FUNCTION_BLOCK CountCurrentPosition1
VAR_INPUT
END_VAR
VAR_OUTPUT
END_VAR
VAR
END_VAR

// COUNT ROTATION:
IF IO.Initialized AND IO.StepRotatonSwitch = 1 THEN
	IF IO.MotorRotationDirection = 0 THEN
		IF (NOT IO.Switch) AND Automatic.RCurrentlyMoving THEN
			IF IO.PreviousManualMode THEN
				Automatic.RotationPositionCurrent := Automatic.RotationPositionCurrent + 1;
			ELSE
				Automatic.RotationPositionCurrent := Automatic.RotationPositionCurrent + 1;
				Automatic.RotationPositionAuto := Automatic.RotationPositionAuto + 1;
			END_IF
		ELSIF Automatic.RCurrentlyMoving THEN
			Automatic.RotationPositionCurrent := Automatic.RotationPositionCurrent + 1;
		END_IF
	ELSE
		IF (NOT IO.Switch) AND Automatic.RCurrentlyMoving THEN
			IF IO.PreviousManualMode THEN
				Automatic.RotationPositionCurrent := Automatic.RotationPositionCurrent - 1;
			ELSE
				Automatic.RotationPositionCurrent := Automatic.RotationPositionCurrent - 1;
				Automatic.RotationPositionAuto := Automatic.RotationPositionAuto - 1;
			END_IF
		ELSIF Automatic.RCurrentlyMoving THEN
			Automatic.RotationPositionCurrent := Automatic.RotationPositionCurrent - 1;
		END_IF
	END_IF
END_IF

// COUNT Extension:
IF IO.Initialized AND IO.StepExtensionSwitch = 1 THEN
	IO.LEDGreen := 0;
	IF IO.MotorExtensionDirection = 0 THEN
		IF (NOT IO.Switch) AND Automatic.ECurrentlyMoving THEN
			IF IO.PreviousManualMode THEN
				Automatic.ExtensionPositionCurrent := Automatic.ExtensionPositionCurrent + 1;
			ELSE
				Automatic.ExtensionPositionAuto := Automatic.ExtensionPositionAuto + 1;
				Automatic.ExtensionPositionCurrent := Automatic.ExtensionPositionCurrent + 1;
			END_IF
		ELSIF Automatic.ECurrentlyMoving THEN
			Automatic.ExtensionPositionCurrent := Automatic.ExtensionPositionCurrent + 1;
		END_IF
	ELSE
		IF (NOT IO.Switch) AND Automatic.ECurrentlyMoving THEN
			IF IO.PreviousManualMode THEN
				Automatic.ExtensionPositionCurrent := Automatic.ExtensionPositionCurrent - 1;
			ELSE
				Automatic.ExtensionPositionAuto := Automatic.ExtensionPositionAuto - 1;
				Automatic.ExtensionPositionCurrent := Automatic.ExtensionPositionCurrent - 1;
			END_IF
		ELSIF Automatic.ECurrentlyMoving THEN
			Automatic.ExtensionPositionCurrent := Automatic.ExtensionPositionCurrent - 1;
		END_IF
	END_IF
END_IF

// COUNT Lifting:
IF IO.Initialized AND IO.StepLiftingSwitch = 1 THEN
	IF IO.MotorLiftingDirection = 0 THEN
		IF (NOT IO.Switch) AND Automatic.LCurrentlyMoving THEN
			IF IO.PreviousManualMode THEN
				Automatic.LiftingPositionCurrent := Automatic.LiftingPositionCurrent + 1;
			ELSE
				Automatic.LiftingPositionCurrent := Automatic.LiftingPositionCurrent + 1;
				Automatic.LiftingPositionAuto := Automatic.LiftingPositionAuto + 1;
			END_IF
		ELSIF Automatic.LCurrentlyMoving THEN
			Automatic.LiftingPositionCurrent := Automatic.LiftingPositionCurrent + 1;
		END_IF
	ELSE
		IF (NOT IO.Switch) AND Automatic.LCurrentlyMoving THEN
			IF IO.PreviousManualMode THEN
				Automatic.LiftingPositionCurrent := Automatic.LiftingPositionCurrent - 1;
			ELSE
				Automatic.LiftingPositionAuto := Automatic.LiftingPositionAuto - 1;
				Automatic.LiftingPositionCurrent := Automatic.LiftingPositionCurrent - 1;
			END_IF
		ELSIF Automatic.LCurrentlyMoving THEN
			Automatic.LiftingPositionCurrent := Automatic.LiftingPositionCurrent - 1;
		END_IF
	END_IF
END_IF

// COUNT Grip:
IF IO.Initialized AND IO.StepGripSwitch = 1 THEN
	IF IO.MotorGripDirection = 0 THEN
		IF (NOT IO.Switch) AND Automatic.GCurrentlyMoving THEN	// automatic mode
			IO.LEDGreen := 0;
			
			IF IO.PreviousManualMode THEN
				Automatic.GripPositionCurrent := Automatic.GripPositionCurrent + 1;
			ELSE
				Automatic.GripPositionAuto := Automatic.GripPositionAuto + 1;
				Automatic.GripPositionCurrent := Automatic.GripPositionCurrent + 1;
			END_IF
		ELSIF Automatic.GCurrentlyMoving THEN		// manual mode
			Automatic.GripPositionCurrent := Automatic.GripPositionCurrent + 1;
		END_IF
	ELSE
		IF (NOT IO.Switch) AND Automatic.GCurrentlyMoving THEN
			IO.LEDGreen := 1;
			IF IO.PreviousManualMode THEN
				Automatic.GripPositionCurrent := Automatic.GripPositionCurrent - 1;
			ELSE
				Automatic.GripPositionAuto := Automatic.GripPositionAuto - 1;
				Automatic.GripPositionCurrent := Automatic.GripPositionCurrent - 1;
			END_IF
		ELSIF Automatic.GCurrentlyMoving THEN
			Automatic.GripPositionCurrent := Automatic.GripPositionCurrent - 1;
		END_IF
	END_IF
END_IF

END_FUNCTION_BLOCK

(* stored: Version 1.1.0.1, ProductVersion 3.1.4024.13
   POU CountCurrentPosition1: Id {9470ef1e-6d57-4400-87bd-bf87707256a6}, SpecialFunc None *)
